// TIA Portal V15.1 export
// export: Created 2024-06-21T08:40:55.6337263Z, ExportSetting WithDefaults, DisplayName Totally Integrated Automation Portal, DisplayVersion V15.1 Update 5, DisplayName TIA Portal Openness, DisplayVersion V15.1 Update 5, DisplayName SINAMICS Startdrive Advanced, DisplayVersion V15.1, DisplayName G130, G150, S120, S150, SINAMICS MV, S210, DisplayVersion V15.1, DisplayName G110M, G120, G120C, G120D, G120P, DisplayVersion V15.1, DisplayName STEP 7 Professional, DisplayVersion V15.1 Update 5, DisplayName STEP 7 Safety, DisplayVersion V15.1, DisplayName WinCC Professional, DisplayVersion V15.1 Update 5, DisplayName SIMATIC Visualization Architect, DisplayVersion V15.1
FUNCTION "LDBCompare" : Void   // FC2101, FBD
TITLE = LDBCompare
{ S7_Optimized_Access := 'FALSE' }
AUTHOR : VCC
FAMILY : Data
VERSION : 0.1
// =============================================================================  This Module Compares Two DB:s  =============================================================================
// stored: AutoNumber false, IsIECCheckEnabled true, SetENOAutomatically False, UDAEnableTagReadback false
   VAR_INPUT
      I_FirstDB : DB_ANY;   // First DB To Check
      I_SecondDB : DB_ANY;   // Startadress Of The First DB
      I_FirstDBStartAdress : Int;   // Second DB To Check
      I_SecondDBStartAdress : Int;   // Startadress Of The Second DB
      I_Length : Word;   // Length To Check
   END_VAR
   VAR_OUTPUT
      O_DBEqual : Bool;   // DB:s Equal
      O_DBNotEqual : Bool;   // DB:s Not Equal
   END_VAR
   VAR_TEMP
      FirstDBCnt : Real;   // First DB Byte
      SecondDBCnt : Real;   // Second DB Byte
      FirstDBByte : Byte;   // Pointer
      SecondDBByte : Byte;   // Pointer
      Length : Real;   // Length
   END_VAR
BEGIN

REGION Network 1: **** 5.2 - Equations - Flow Equations **** DB:s Not Equal
   // DB:s Not Equal
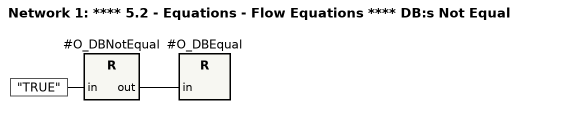
   IF "TRUE" THEN
       #O_DBNotEqual := FALSE;
       #O_DBEqual := FALSE;
   END_IF;
END_REGION

NETWORK
TITLE = **** 5.2 - Equations - Flow Equations **** Load Pointers
// Load Pointers

//APA Fixa,
      L     #I_FirstDBStartAdress;
      L     P#1.0;
      *I;
      T     #FirstDBCnt;
      L     #I_SecondDBStartAdress;
      L     P#1.0;
      *I;
      T     #SecondDBCnt;

Again:OPN   #I_FirstDB;
      L     DBB [#FirstDBCnt];
      T     #FirstDBByte;

      OPN   #I_SecondDB;
      L     DBB [#SecondDBCnt];
      T     #SecondDBByte;

      A(;

      L     #FirstDBByte;
      L     #SecondDBByte;

      <>I;

      );

      S     #O_DBNotEqual;
      R     #O_DBEqual;

      JC    End;

      L     #FirstDBCnt;
      L     P#1.0;
      +I;
      T     #FirstDBCnt;

      L     #SecondDBCnt;
      L     P#1.0;
      +I;
      T     #SecondDBCnt;

      L     #I_Length;
      L     #I_FirstDBStartAdress;
      +I;
      L     P#1.0;
      *I;
      L     P#1.0;
      -I;
      T     #Length;

      A(;

      L     #FirstDBCnt;
      L     #Length;
      >I;

      );

      R     #O_DBNotEqual;
      S     #O_DBEqual;
      JC    End;
      JU    Again;
End:  NOP   0;



END_FUNCTION
